(* CODESYS project intecreutilities.library
   DocFormat: reStructuredText
   Company: Intecre Ltd
   DefaultNamespace: Intecre.Utilities
   Title: Intecre.Utilities
   Placeholder: Intecre.Utilities
   Author: Mark Lazarides
   Description: 3.1.1.0 - adding long string list
      
      3.1.0.0 
      - Adding external logging injection
      3.0.0.0 
      - Renamed TNamedBase to T_NamedBase 
      - Added NONE level logging.
      - Logging is "NONE" by default.
      - Use something like "Intecre_Utilities.LogConfig.LogLevel := E_LogSeverity.Error; " to turn all on.
   Version: 3.1.1.0

Project tree, tasks and I/O mapping:
  libraries: Tc2_Math, * (Beckhoff Automation GmbH); Tc2_MDP, * (Beckhoff Automation GmbH); Tc2_Standard, * (Beckhoff Automation GmbH); Tc2_System, * (Beckhoff Automation GmbH); Tc2_Utilities, * (Beckhoff Automation GmbH); Tc3_Module, * (Beckhoff Automation GmbH)
  DUTs/
  GVLs/
    global variables CollectionParameters
    global variables LogConfig
    global variables Objects
    global variables StringsParams
  Project Information/
    function F_GetCompany [ST]
    function F_GetTitle [ST]
    function F_GetVersion [ST]
  System/
    function block T_Task [ST]: CycleCount, CyclesPerSecond, CycleTimeExceeded, CycleTimeInMs, CycleTimeInSecs, DateString, DateTimeFromDc, DateTimeString, DistributedClockTimeInMs, DistributedClockTimeInNs, DistributedClockTimeInSecs, Index, IsFirstScan, Name, TimeString, SetToThisTask
  Terminal Interfaces/
    Analogue Input EL3xxx/
      EL3058/
        data type stEL3058_Channel
        data type stEL3058_ChannelStatus
      EL3152/
        data type stEL3152_Channel
        data type stEL3152_ChannelStatus
      EL3318/
        data type stEL3318_Channel
        data type stEL3318_ChannelStatus
    EtherCAT Standard/
      data type stInfoData
      data type stWcState
    System EL9xxx/
      EL9410/
        data type stEL9410
      EL9576/
        data type stEL9576
        data type stEL9576_Status
  Utilities/
    Conversion/
      function CharIsNumber [ST]
      function CharIsNumberOrPeriod [ST]
      function TryStringToLreal [ST]
      function TryStringToUdint [ST]
      function TryStringToWord [ST]
    IPC Diagnostics/
      function block T_MdpReadCpuTemp [ST]: Busy, CpuTemp, Error, ErrorId, SetUpdateTimerValue
    Logger/
      data type E_LogSeverity
      function F_LogDebug [ST]
      function F_LogError [ST]
      function F_Logger [ST]
      function F_LogInfo [ST]
      function F_LogWarning [ST]
      function block FB_LogErrorEdge [ST]
      function block FB_LogInfoEdge [ST]
      function block FB_LogOnEdge [ST]
      function block FB_LogWarningEdge [ST]
      interface I_ExternalLogger: AddToLog
    Object Tracking/
      function F_DictionaryValuesCrc [ST]
      function block FB_Dictionary [ST]: AddItem, Clear, Contains, Count, Get, ReferenceToThis, Remove, TryGet, TryGetIndex, TryGetPartialKey
      function block FB_PointerList [ST]: AddItem, Clear, Contains, Count, FindIndex, GetIndex, RemoveIndex, TryGetIndex
      function block FB_StringList [ST]: AddItem, Clear, Contains, ContainsPartial, CopyList, CopyListAndClear, Count, FindIndex, FindIndexPartialKey, GetIndex, RemoveIndex, TryGetIndex
      function block FB_LongStringList [ST]: AddItem, Clear, Contains, ContainsPartial, CopyList, CopyListAndClear, Count, FindIndex, FindIndexPartialKey, GetIndex, RemoveIndex, TryGetIndex
      function block FB_TargList [ST]: AddItem, Clear, Contains, Count, FindIndex, GetIndex, RemoveIndex, TryGetIndex
      function block FB_UdintList [ST]: AddItem, Clear, Contains, Count, FindIndex, GetIndex, RemoveIndex, TryGetIndex
      global variables GVL_List
      data type ST_KeyReferencePair
    PI Controller/
      function block FB_I_Controller [ST]
      function block FB_P_Control [ST]
      function block FB_PI_Controller [ST]
    String/
      Large Concats/
        function F_ClearLarge [ST]
        function F_Concat3_Large [ST]
        function F_Concat4_Large [ST]
        function F_Concat5_Large [ST]
        function F_Concat6_Large [ST]
        function F_Concat7_Large [ST]
        function F_ConcatLarge [ST]
      data type LongString
      function F_Concat3 [ST]
      function F_Concat4 [ST]
      function F_Concat5 [ST]
      function F_Concat6 [ST]
      function F_Concat7 [ST]
      function F_StringToTarg [ST]
      function F_TargToString [ST]
    Testing/
      function block FB_Assert [ST]: FinishedTestingMsg, FloatsAreDifferent, FloatsAreEqual, IsFalse, IsTrue, StartTestingMsg
      function block T_TestBase [ST]: Done, DonePulse, nElapsedTimeInMs, Passed, Reset, Start, StartTimer, tElapsedTimeInMs
    Timers/
      function block T_Timer [ST]: ElapsedTime, ElapsedTimeInMs, Q_Off, Q_On, Q_PulseTrain, SetPeriod, Signal
    Write persistent/
      function block T_WritePersistentData [ST]: SetConfig
    function F_Gate [ST]
    function block T_NamedBase [ST]: InstanceName, LogDebug, LogError, LogInfo, LogWarning, setInstanceName
  Version/
    global variables Global_Version
  VISUs/
*)

// Terminal Interfaces/Analogue Input EL3xxx/EL3058/stEL3058_Channel
{attribute 'pack_mode' := '1'}
TYPE stEL3058_Channel :
STRUCT
	Status	AT %I* : stEL3058_ChannelStatus;
	Value 	AT %I* : WORD;
END_STRUCT
END_TYPE

// Terminal Interfaces/Analogue Input EL3xxx/EL3058/stEL3058_ChannelStatus
TYPE stEL3058_ChannelStatus :
STRUCT
	Underrange 	: BIT;
	Overrange	: BIT;
	Limit1_0	: BIT; // Value <= limit 1
	Limit1_1 	: BIT; // Value >= limit 1
	Limit2_0	: BIT; // Value <= limit 2
	Limit2_1	: BIT; // Value >= limit 2
	Error		: BIT; // TRUE when Over or under range.
	{attribute 'hide'}
	padding_0_7	: BIT;
	{attribute 'hide'}
	padding_1_0 : BIT;
	{attribute 'hide'}
	padding_1_1 : BIT;
	{attribute 'hide'}
	padding_1_2 : BIT;
	{attribute 'hide'}
	padding_1_3 : BIT;
	{attribute 'hide'}
	padding_1_4 : BIT;
	{attribute 'hide'}
	padding_1_5 : BIT;
	TxPDO_State : BIT; // TRUE when PDO NOT valid
	TxPDO_Toddle: BIT; // toggles when new value available
END_STRUCT
END_TYPE

// Terminal Interfaces/Analogue Input EL3xxx/EL3152/stEL3152_Channel
{attribute 'pack_mode' := '1'}
TYPE stEL3152_Channel:
STRUCT
	Status 	AT %I* : stEL3152_ChannelStatus;	
	Value 	AT %I* : WORD;  
END_STRUCT
END_TYPE;

// Terminal Interfaces/Analogue Input EL3xxx/EL3152/stEL3152_ChannelStatus
{attribute 'pack_mode' := '1'}
TYPE stEL3152_ChannelStatus:
STRUCT
	Underrange 	: BIT;
	Overrange 	: BIT;
	LT_Lim1 	: BIT; // Less Than Limit 1
	GT_Lim1 	: BIT; // Greater Than Limit 1
	LT_Lim2 	: BIT; // Less Than Limit 2
	GT_Lim2 	: BIT; // Greater Than Limit 2
	Error		: BIT;
	{attribute 'hide'}
	pack0_7		: BIT;	
	{attribute 'hide'}
	pack1_0		: BIT;
	{attribute 'hide'}
	pack1_1	 	: BIT;
	{attribute 'hide'}
	pack1_2	 	: BIT;
	{attribute 'hide'}
	pack1_3	 	: BIT;
	{attribute 'hide'}
	pack1_4	 	: BIT;
	SyncError	: BIT;
	TxPDOState	: BIT;
	TxPDOToggle : BIT;
END_STRUCT
END_TYPE;

// Terminal Interfaces/Analogue Input EL3xxx/EL3318/stEL3318_Channel
{attribute 'pack_mode' := '2'}
TYPE stEL3318_Channel:
STRUCT
	Status 	AT %I* : stEL3318_ChannelStatus;	 
	Value 	AT %I* : WORD;  
END_STRUCT
END_TYPE;

// Terminal Interfaces/Analogue Input EL3xxx/EL3318/stEL3318_ChannelStatus
{attribute 'pack_mode' := '1'}
TYPE stEL3318_ChannelStatus:
STRUCT
	Underrange 	: BIT;
	Overrange 	: BIT;
	{attribute 'hide'}
	pack_0_2	: BIT;
	{attribute 'hide'}
	pack_0_3	: BIT;
	{attribute 'hide'}
	pack_0_4	: BIT;
	{attribute 'hide'}
	pack_0_5	: BIT;
	Error		: BIT;
	{attribute 'hide'}	
	pack_0_7	: BIT;
	{attribute 'hide'}
	pack_1_0 	: BIT;
	{attribute 'hide'}
	pack_1_1 	: BIT;
	{attribute 'hide'}
	pack_1_2	: BIT;
	{attribute 'hide'}
	pack_1_3	: BIT;
	{attribute 'hide'}
	pack_1_4	: BIT;
	{attribute 'hide'}
	pack_1_5	: BIT;
	TxPDOState	: BIT;
	TxPDOToggle : BIT;

END_STRUCT
END_TYPE;

// Terminal Interfaces/EtherCAT Standard/stInfoData
TYPE stInfoData :
STRUCT
	State 		AT %I* : WORD;
	InfoData 	AT %I* : AMSADDR;
END_STRUCT
END_TYPE

// Terminal Interfaces/EtherCAT Standard/stWcState
TYPE stWcState :
STRUCT
	WcState		AT %I* : BOOL; // FALSE = data valid, TRUE = data not valid
	InputToggle	AT %I* : BOOL; // toggles every scan.
END_STRUCT
END_TYPE

// Terminal Interfaces/System EL9xxx/EL9410/stEL9410
TYPE stEL9410 :
STRUCT
	Us_Undervoltage  AT%I* : BIT; 
	Up_Undervoltage AT %I* : BIT; 
END_STRUCT
END_TYPE

// Terminal Interfaces/System EL9xxx/EL9576/stEL9576
{attribute 'pack_mode' := '1'}
TYPE stEL9576 :
STRUCT
	BCT_Inputs AT %I* : stEL9576_Status; 
END_STRUCT
END_TYPE;

// Terminal Interfaces/System EL9xxx/EL9576/stEL9576_Status
{attribute 'pack_mode' := '1'}
TYPE stEL9576_Status :
STRUCT
	TermOvertemp 	: BIT;
	I2T_Err 		: BIT;
	I2T_Warning 	: BIT; 
	Overvoltage 	: BIT; 
	Undervoltage 	: BIT; 
	ChopperOn 		: BIT;
	{attribute 'hide'}
	pack0_6		: BIT;
	{attribute 'hide'}
	pack0_7		: BIT;
	{attribute 'hide'}
	pack1_0		: BIT;
	{attribute 'hide'}
	pack1_1	 	: BIT;
	{attribute 'hide'}
	pack1_2	 	: BIT;
	{attribute 'hide'}
	pack1_3	 	: BIT;
	{attribute 'hide'}
	pack1_4	 	: BIT;
	{attribute 'hide'}
	pack1_5	 	: BIT;
	InputCycCnt_0	: BIT;
	InputCycCnt_1	: BIT;
	DcLinkVoltage	: UDINT;
	ResistorCurrent	: DINT;
	DutyCycle 		: USINT;
	I2T_LoadFactor 	: USINT;
END_STRUCT
END_TYPE;

// Utilities/Logger/E_LogSeverity
{attribute 'qualified_only'}
TYPE E_LogSeverity :
(
	Debug := 0,
	Info := ADSLOG_MSGTYPE_HINT,
	Warning := ADSLOG_MSGTYPE_WARN,
	Error := ADSLOG_MSGTYPE_ERROR,
	None := 1000
) DWORD;
END_TYPE

// Utilities/Object Tracking/ST_KeyReferencePair
TYPE ST_KeyReferencePair :
STRUCT
	Key : T_MaxString;
	Ref : T_Arg;
END_STRUCT
END_TYPE

// Utilities/String/LongString
TYPE LongString : STRING(StringsParams.MAX_STRING_LENGTH); END_TYPE // use StringsParams.MAX_STRING_LENGTH to adjust length

// GVLs/CollectionParameters
{attribute 'qualified_only'}
VAR_GLOBAL CONSTANT
	MAX_BYTE_SIZE : UDINT := 1000;
END_VAR

// GVLs/LogConfig
{attribute 'qualified_only'}
VAR_GLOBAL
	// set level to log. Lower log level includes higher levels i.e. info does warning and Error. 
	LogLevel : E_LogSeverity := E_LogSeverity.None; // Turn messages off by default
	ExternalLogger : I_ExternalLogger; // permit logging to something else
END_VAR

// GVLs/Objects
{attribute 'qualified_only'}
{attribute 'strict'}
VAR_GLOBAL 
	
END_VAR

// GVLs/StringsParams
{attribute 'qualified_only'}
VAR_GLOBAL CONSTANT
	MAX_STRING_LENGTH : UDINT := 300; // used for all string concats.
END_VAR

// Utilities/Object Tracking/GVL_List
{attribute 'qualified_only'}
VAR_GLOBAL CONSTANT
	LIST_SIZE : UINT := 100; // Number of list items.
END_VAR

// Version/Global_Version
{attribute 'TcGenerated'}
{attribute 'no-analysis'}
{attribute 'linkalways'}
// This function has been automatically generated from the project information.
VAR_GLOBAL CONSTANT
	{attribute 'const_non_replaced'}
	stLibVersion_Intecre_Utilities : ST_LibVersion := (iMajor := 3, iMinor := 1, iBuild := 1, iRevision := 0, sVersion := '3.1.1.0');
END_VAR

// Project Information/F_GetCompany
// This function has been automatically generated from the project information.
{attribute 'signature_flag' := '1073741824'}
{attribute 'TcGenerated'}
{attribute 'no-analysis'}
FUNCTION F_GetCompany : WSTRING
VAR_INPUT
	
END_VAR

F_GetCompany := "Intecre Ltd";

END_FUNCTION

// Project Information/F_GetTitle
// This function has been automatically generated from the project information.
{attribute 'signature_flag' := '1073741824'}
{attribute 'TcGenerated'}
{attribute 'no-analysis'}
FUNCTION F_GetTitle : WSTRING
VAR_INPUT
	
END_VAR

F_GetTitle := "Intecre.Utilities";

END_FUNCTION

// Project Information/F_GetVersion
// This function has been automatically generated from the project information.
{attribute 'signature_flag' := '1073741824'}
{attribute 'TcGenerated'}
{attribute 'no-analysis'}
FUNCTION F_GetVersion : ST_LibVersion
VAR_INPUT
	
END_VAR

F_GetVersion.iMajor := 3;
F_GetVersion.iMinor := 1;
F_GetVersion.iBuild := 1;
F_GetVersion.iRevision := 0;

END_FUNCTION

// System/T_Task
// Exposes _TaskInfo[x] information for the task index the object is instantied in.
//
// After declaration, each property can be directly accessed.
//
// Set the index using task.Index
FUNCTION_BLOCK T_Task // Simply exposes task information.
VAR
// Backing Properties
	_index : BYTE := 1;
	_cycleTimeInMs : LREAL;
	_isFirstScan : BOOL;
	_cycleTimeExceeded : BOOL;
	_name : STRING(63);
	_runTimeInMs : UDINT;
	_distributedClockTimeInMs : LINT;
	_distributedClockTimeInNs : LINT;

// FBs
	initialised : BOOL := FALSE;
	taskIndex : GETCURTASKINDEX;
	
END_VAR

VAR CONSTANT
	HUNDRED_NS_IN_MS : LINT := 10000;
	NS_IN_MS : LINT := 1000000;
END_VAR

// Number of task cycles executed.
PROPERTY PUBLIC CycleCount : UDINT
GET
cycleCount := TwinCAT_SystemInfoVarList._TaskInfo[_index].CycleCount;
END_GET
END_PROPERTY

// Configured cycles per second (1 / task time)
PROPERTY CyclesPerSecond : LREAL
GET
CyclesPerSecond := 1 / CycleTimeInSecs;
END_GET
END_PROPERTY

// Last cycle time exceeded
PROPERTY CycleTimeExceeded : BOOL
GET
_cycleTimeExceeded := TwinCAT_SystemInfoVarList._TaskInfo[_index].CycleTimeExceeded;
cycleTimeExceeded := _cycleTimeExceeded;
END_GET
END_PROPERTY

// Configured task cycle time in ms
PROPERTY CycleTimeInMs : LREAL
GET
_cycleTimeInMs := TwinCAT_SystemInfoVarList._TaskInfo[_index].CycleTime / LINT_TO_UDINT(HUNDRED_NS_IN_MS); // CycleTime expressed in 100ns units.
cycleTimeInMs := _cycleTimeInMs;
END_GET
END_PROPERTY

// Configured task cycle time in seconds
PROPERTY CycleTimeInSecs : LREAL
GET
CycleTimeInSecs:= CycleTimeInMs / 1000;
END_GET
END_PROPERTY

PROPERTY DateString : STRING
GET
VAR
	temp : STRING;
END_VAR
// remove the trailing time: 2018-07-30_09-23-47
temp := DELETE( TO_STRING( DateTimeString ), 9,11 );

// 2018-07-30
DateString :=  temp;
END_GET
END_PROPERTY

PROPERTY DateTimeFromDc : DATE_AND_TIME
GET
DateTimeFromDc := LINT_TO_DT( TO_LINT( DT#2000-1-1-00:00 ) + TwinCAT_SystemInfoVarList._TaskInfo[_index].DcTaskTime / 1000000000 );
END_GET
END_PROPERTY

PROPERTY DateTimeString : STRING
GET
VAR
	temp : STRING;
END_VAR
// remove the leading DT# : DT#2018-07-30-09:23:47
temp := DELETE( TO_STRING( DateTimeFromDc ), 3, 1 );
// add underscore between datae and time 2018-07-30-09:23:47
temp := REPLACE( temp, '_', 1, 11 );
// replace the colons with dashes 2018-07-30_09:23:47
temp := REPLACE( REPLACE( temp, '-', 1, 14 ), '-', 1, 17 );

// 2018-07-30_09-23-47
DateTimeString :=  temp;
END_GET
END_PROPERTY

//Distributed clock time in milliseconds.
PROPERTY PUBLIC DistributedClockTimeInMs : LINT
GET
_distributedClockTimeInMs := TwinCAT_SystemInfoVarList._TaskInfo[_index].DcTaskTime / NS_IN_MS; // CycleTime expressed ns.
DistributedClockTimeInMs := _distributedClockTimeInMs;
END_GET
END_PROPERTY

//Distributed clock time in nanoseconds.
PROPERTY PUBLIC DistributedClockTimeInNs : LINT
GET
_distributedClockTimeInNs := TwinCAT_SystemInfoVarList._TaskInfo[_index].DcTaskTime; // CycleTime expressed ns.
DistributedClockTimeInNs := _distributedClockTimeInNs;
END_GET
END_PROPERTY

//Distributed clock time in milliseconds.
PROPERTY PUBLIC DistributedClockTimeInSecs : LINT
GET
DistributedClockTimeInSecs := DistributedClockTimeInMs / 1000;
END_GET
END_PROPERTY

//Get/Set the task for the infomration required. Can use "SetToThisTask()" to set to local task.
PROPERTY PUBLIC Index : BYTE
GET
PUBLIC
Index := _index;
END_GET
SET
PUBLIC
_index := Index;
END_SET
END_PROPERTY

PROPERTY IsFirstScan : BOOL
GET
_isFirstScan := TwinCAT_SystemInfoVarList._TaskInfo[_index].FirstCycle;
IsFirstScan := _isFirstScan;
END_GET
END_PROPERTY

{attribute 'monitoring' := 'call'}
PROPERTY Name : STRING(63)
GET
_name := TwinCAT_SystemInfoVarList._TaskInfo[_index].TaskName;
Name := _name;
END_GET
END_PROPERTY

PROPERTY TimeString : STRING
GET
VAR
	temp : STRING;
END_VAR
// remove the leading date 2018-07-30_09-23-47
temp := DELETE( TO_STRING( DateTimeString ), 11, 1 );

// 09-23-47
TimeString :=  temp;
END_GET
END_PROPERTY

//set the task object to this task
METHOD PUBLIC SetToThisTask : BOOL
VAR
	curTask : GETCURTASKINDEX;
END_VAR
curTask();
Index := curTask.index;
END_METHOD

END_FUNCTION_BLOCK

// Utilities/Conversion/CharIsNumber
FUNCTION CharIsNumber : BOOL
VAR_INPUT
	bChar : BYTE; // char to check
END_VAR

// check bChar is in numbr range of ascii
CharIsNumber := (bChar >= 48 AND bChar <=57);

END_FUNCTION

// Utilities/Conversion/CharIsNumberOrPeriod
FUNCTION CharIsNumberOrPeriod : BOOL
VAR_INPUT
	bChar : BYTE; // char to check
END_VAR

// check is bChar in number range of ascii, or a period (full-stop).
CharIsNumberOrPeriod := CharIsNumber( bChar ) OR_ELSE (bChar = 46);

END_FUNCTION

// Utilities/Conversion/TryStringToLreal
// Returns TRUE if possible. sVal will hold value if passes.
FUNCTION TryStringToLreal : BOOL 
VAR_INPUT
	sStringToParse : STRING; // String to try
END_VAR
VAR_IN_OUT
	sVal : LREAL; // 0.0 (zero) if fails, parsed value if passes.
END_VAR
VAR
	i : INT;
	n : INT; // position of full stop (if at all).
	intPart : DINT; // integer part of the number.
	decPart : UDINT; // decimal part of the number.
	decPartAsLreal : LREAL;
	decimalPlaces : INT; // number of dps.
	isMinus : BOOL;
END_VAR

IF LEN(sStringToParse) > 0 THEN

	FOR i := 0 TO LEN(sStringToParse) - 1 DO	
		
		IF i = 0 AND_THEN sStringToParse[i] = 45 THEN // accept "minus" sign for first digit
			isMinus := TRUE;
		ELSIF i = 1 AND isMinus THEN // if first char is "-", second must be digit.
			IF NOT CharIsNumberOrPeriod( sStringToParse[i] ) THEN
				sVal := 0;
				RETURN;
			END_IF
		ELSIF NOT CharIsNumberOrPeriod( sStringToParse[i] ) THEN
			sVal := 0;
			RETURN;
		END_IF	
	END_FOR
	
	n := FIND(sStringToParse, '.');
	
	IF n > 0 THEN // full stop is in the string.
		// get integer part.
		intPart := STRING_TO_DINT(LEFT(sStringToParse, n - 1));
		decimalPlaces := LEN(sStringToParse) - n;
		// get decimal part as integer.
		decPart := STRING_TO_UDINT( RIGHT(sStringToParse, decimalPlaces) );
		// convert to LREAL, includng rolling decimal places.
		decPartAsLreal := UDINT_TO_LREAL(decPart)/EXPT(10,decimalPlaces);
		// handle sign change.
		IF isMinus THEN
			decPartAsLreal := decPartAsLreal * -1;
		END_IF
		
		//combine them
		sVal := DINT_TO_LREAL(intPart);
		sVal := sVal + decPartAsLreal;
	ELSE
		sVal := STRING_TO_LREAL(sStringToParse);
	END_IF
	
	TryStringToLreal := TRUE;
	
END_IF

END_FUNCTION

// Utilities/Conversion/TryStringToUdint
// Returns TRUE if possible. sVal will hold value if passes.
FUNCTION TryStringToUdint : BOOL 
VAR_INPUT
	sStringToParse : STRING; // String to try
END_VAR
VAR_IN_OUT
	sVal : UDINT; // 0 (zero) if fails, parsed value if passes.
END_VAR
VAR
	i : INT;
END_VAR

IF LEN(sStringToParse) > 0 THEN

	FOR i := 0 TO LEN(sStringToParse) - 1 DO		
		IF NOT CharIsNumber( sStringToParse[i] ) THEN
			sVal := 0;
			RETURN;
		END_IF	
	END_FOR
	
	sVal := STRING_TO_UDINT( sStringToParse );
	TryStringToUdint := TRUE;
	
END_IF

END_FUNCTION

// Utilities/Conversion/TryStringToWord
// Returns TRUE if possible. sVal will hold value if passes. 
//
// Internally this casts to Udint, then checks value is <= MAX_WORD
FUNCTION TryStringToWord : BOOL 
VAR_INPUT
	sStringToParse : STRING; // String to try
END_VAR
VAR_IN_OUT
	sVal : WORD; // 0 (zero) if fails, parsed value if passes.
END_VAR
VAR
	u : UDINT;
END_VAR

// check parsing to UDINT possible, then validate size of word.
IF TryStringToUdint(sStringToParse, u) THEN
	// check within WORD size.
	IF UDINT_TO_WORD(u) <= 65535 THEN
		sVal := STRING_TO_WORD( sStringToParse );
		TryStringToWord := TRUE;
	END_IF
	
END_IF

END_FUNCTION

// Utilities/IPC Diagnostics/T_MdpReadCpuTemp
/// cyclically reads the  cpu temp at specified update period. Default is 500ms.
{attribute 'contains_implicit_enum'}
FUNCTION_BLOCK T_MdpReadCpuTemp
VAR
	/// local read                
	amsNetId: STRING := '';
	mdpAddr: ST_MDP_Addr;
	updateTimer: TON := (PT := TIME#500ms);
	readMdpElement: FB_MDP_ReadElement;
	/// returned from MDP read element 
	rawData: UINT;
	_cpuTemp: INT;
	{attribute 'implicit_enum_type' := ''}
	state:(
		mrctInit  := 0,     // initiate state machine (set parameters)
		mrctReadCpuTemp,
		mrctWaitForReadComplete,
		mrctProcessCpuTemp
	);   
END_VAR
VAR CONSTANT
	/// from IPC Diagnostics Manual V1.8, p63 
	CPU_PROPERTIES_TABLE_NUMBER: BYTE := 1;
	/// from IPC Diagnostics Manual V1.8, p63 
	CPU_TEMP_SUB_INDEX_OF_CPU_PROPS_TABLE: BYTE := 3;
END_VAR

CASE state OF

	mrctInit : 
		
		// timer starts the read process.
		state := 
			SEL ( updateTimer.Q, state, mrctReadCpuTemp );
		
	mrctReadCpuTemp :    
      
		state := mrctWaitForReadComplete;  
            
	mrctWaitForReadComplete :    

		IF NOT readMdpElement.bBusy THEN
			
			state := mrctProcessCpuTemp;
			
		END_IF
	
	mrctProcessCpuTemp :              

		IF NOT readMdpElement.bError THEN
			MEMCPY( ADR( _cpuTemp ), ADR( rawData ), SIZEOF( rawData ) );
			
		END_IF
		
		state    := mrctInit; 
		
ELSE
	
    state := mrctInit;   
	 
END_CASE 

updateTimer( 
	IN := state = mrctInit
);
		
mdpAddr.nArea := INT_TO_BYTE(eMDP_Area_ConfigArea); 
mdpAddr.nTableId := CPU_PROPERTIES_TABLE_NUMBER;            
mdpAddr.nSubIdx := CPU_TEMP_SUB_INDEX_OF_CPU_PROPS_TABLE;   

readMdpElement(
	bExecute	:= state = mrctReadCpuTemp,               
	eModuleType	:= E_MDP_ModuleType.eMDP_ModT_CPU,         
	stMDP_Addr := mdpAddr,          
	iModIdx := 0,                   
	pDstBuf := ADR(rawData),         
	cbDstBufLen := SIZEOF(rawData),  
	sAmsNetId := amsNetId,        
);

{attribute 'monitoring' := 'variable'}
PROPERTY Busy : BOOL
GET
Busy := state <> mrctInit;
END_GET
END_PROPERTY

{attribute 'monitoring' := 'call'}
PROPERTY CpuTemp : INT
GET
CpuTemp := THIS^._cpuTemp;
END_GET
END_PROPERTY

{attribute 'monitoring' := 'variable'}
PROPERTY Error : BOOL
GET
Error := NOT Busy AND readMdpElement.bError;
END_GET
END_PROPERTY

{attribute 'monitoring' := 'variable'}
PROPERTY ErrorId : UDINT
GET
ErrorId := SEL( Busy, readMdpElement.nErrID, 0 );
END_GET
END_PROPERTY

METHOD SetUpdateTimerValue 
VAR_INPUT	
	UpdatePeriod: TIME;
END_VAR
IF UpdatePeriod > T#1MS THEN
	THIS^.updateTimer.PT := UpdatePeriod;
END_IF
END_METHOD

END_FUNCTION_BLOCK

// Utilities/Logger/F_LogDebug
FUNCTION F_LogDebug : STRING;
VAR_INPUT
	Message : T_MaxString;
END_VAR

F_LogDebug := 
	F_Logger( 
		E_LogSeverity.Debug, 
		CONCAT( 'DEBUG ' , Message ) 
	);

END_FUNCTION

// Utilities/Logger/F_Logger
FUNCTION F_Logger : STRING;
VAR_INPUT
	LogSeverity : E_LogSeverity;
	Message : T_MaxString;
END_VAR

IF ( LogSeverity < E_LogSeverity.None ) 
	AND_THEN ( LogSeverity >= LogConfig.LogLevel ) THEN
	
	ADSLOGSTR(LogSeverity OR ADSLOG_MSGTYPE_LOG, Message, '');
	F_Logger := Message;
	
	IF LogConfig.ExternalLogger <> 0 THEN
		LogConfig.ExternalLogger.AddToLog( Message, LogSeverity );
	END_IF
	
END_IF

END_FUNCTION

// Utilities/Logger/F_LogError
FUNCTION F_LogError : STRING;
VAR_INPUT
	Message : T_MaxString;
END_VAR

F_LogError := F_Logger(ADSLOG_MSGTYPE_ERROR, Message);

END_FUNCTION

// Utilities/Logger/F_LogInfo
FUNCTION F_LogInfo : STRING;
VAR_INPUT
	Message : T_MaxString;
END_VAR

F_LogInfo := F_Logger(ADSLOG_MSGTYPE_HINT, Message);

END_FUNCTION

// Utilities/Logger/F_LogWarning
FUNCTION F_LogWarning : STRING;
VAR_INPUT
	Message : T_MaxString;
END_VAR

F_LogWarning := F_Logger(ADSLOG_MSGTYPE_WARN, Message);

END_FUNCTION

// Utilities/Logger/FB_LogErrorEdge
FUNCTION_BLOCK FB_LogErrorEdge
VAR_INPUT
	Event : BOOL; // Event flag
	Message : T_MaxString; // Log message
	EventFallingEdge : BOOL := FALSE; // Defined which edge: FALSE = rising TRUE = falling, 
END_VAR
VAR_OUTPUT
	Q : BOOL;
END_VAR
VAR
	fbLogEdge : FB_LogOnEdge;
END_VAR

fbLogEdge(
	Event:= Event, 
	Message:= Message, 
	LogSeverity:= E_LogSeverity.Error, 
	EventFallingEdge:= EventFallingEdge,
	Q => Q
);

END_FUNCTION_BLOCK

// Utilities/Logger/FB_LogOnEdge
FUNCTION_BLOCK FB_LogOnEdge
VAR_INPUT
	Event : BOOL; // look for edge here to log.
	Message : T_MaxString; // message
	LogSeverity : E_LogSeverity; // severity
	EventFallingEdge : BOOL := FALSE; // TRUE for falling edge, FALSE for rising edge.
END_VAR
VAR_OUTPUT
	Q : BOOL;
END_VAR
VAR
	rt : R_TRIG;
	ft : F_TRIG;
END_VAR
VAR_TEMP
	logNow : BOOL;
END_VAR

rt(CLK := Event);
ft(CLK := Event);

Q := SEL(EventFallingEdge, rt.Q, ft.Q);

IF Q THEN
	
	CASE LogSeverity OF
		
		E_LogSeverity.Info : F_LogInfo(Message);
			
		E_LogSeverity.Warning :	F_LogWarning(Message);
			
		E_LogSeverity.Error : F_LogError(Message);
	ELSE 
		
		F_LogError(
			CONCAT(
				'Error in FB_LogOnEdge, Logseverity incorrect. Log Message for event is : ', 
				Message
			)
		);
		
	END_CASE
	
END_IF

END_FUNCTION_BLOCK

// Utilities/Logger/FB_LogInfoEdge
FUNCTION_BLOCK FB_LogInfoEdge
VAR_INPUT
	Event : BOOL; // Event flag
	Message : T_MaxString; // Log message
	EventFallingEdge : BOOL := FALSE; // Defined which edge: FALSE = rising TRUE = falling, 
END_VAR
VAR_OUTPUT
	Q : BOOL;
END_VAR
VAR
	fbLogEdge : FB_LogOnEdge;
END_VAR

fbLogEdge(
	Event:= Event, 
	Message:= Message, 
	LogSeverity:= E_LogSeverity.Info, 
	EventFallingEdge:= EventFallingEdge,
	Q => Q
);

END_FUNCTION_BLOCK

// Utilities/Logger/FB_LogWarningEdge
FUNCTION_BLOCK FB_LogWarningEdge
VAR_INPUT
	Event : BOOL; // Event flag
	Message : T_MaxString; // Log message
	EventFallingEdge : BOOL := FALSE; // Defined which edge: FALSE = rising TRUE = falling, 
END_VAR
VAR_OUTPUT
	Q : BOOL;
END_VAR
VAR
	fbLogEdge : FB_LogOnEdge;
END_VAR

fbLogEdge(
	Event:= Event, 
	Message:= Message, 
	LogSeverity:= E_LogSeverity.Warning, 
	EventFallingEdge:= EventFallingEdge,
	Q => Q
);

END_FUNCTION_BLOCK

// Utilities/Logger/I_ExternalLogger
INTERFACE I_ExternalLogger

METHOD AddToLog
VAR_IN_OUT
	Message : T_MaxString;
END_VAR
VAR_INPUT
	LogSeverity : E_LogSeverity;
END_VAR
END_METHOD

END_INTERFACE

// Utilities/Object Tracking/F_DictionaryValuesCrc
// Return CRC of the values stored in the dictionary.
FUNCTION F_DictionaryValuesCrc : WORD
VAR_IN_OUT
	Dictionary : FB_Dictionary;
END_VAR
VAR
	i : UDINT;
	sKey : T_MaxString;
	tValue : T_Arg;
END_VAR

IF Dictionary.Count > 0 THEN
	
	IF NOT Dictionary.TryGetIndex(Index := 0, Key := sKey, Value := tValue) THEN
		RETURN;
	ELSE
		F_DictionaryValuesCrc := F_DATA_TO_CRC16_CCITT(
			pData := tValue.pData,
			cbData := tValue.cbLen,
			crc := 16#FFFF // First pass needs the seed.
			);
	END_IF
	
END_IF

FOR i := 1 TO (Dictionary.Count -1) DO
	
	IF NOT Dictionary.TryGetIndex(Index := 0, Key := sKey, Value := tValue) THEN
		F_DictionaryValuesCrc := 16#0000;
		RETURN;
	ELSE
		F_DictionaryValuesCrc := F_DATA_TO_CRC16_CCITT(
			pData := tValue.pData,
			cbData := tValue.cbLen,
			crc := F_DictionaryValuesCrc // iteratively pass in CRC.
			);
	END_IF
	
END_FOR

END_FUNCTION

// Utilities/Object Tracking/FB_Dictionary
FUNCTION_BLOCK FB_Dictionary EXTENDS T_NamedBase
VAR
	Keys : FB_StringList;
	Values : FB_TargList;
END_VAR

// Add item to list. TRUE if successful. 
METHOD PUBLIC AddItem : BOOL
VAR_INPUT
	Key : T_MaxString; // item key to add.
	Value : T_Arg;
END_VAR
IF Keys.Count <> Values.Count THEN
	LogWarning('Missmatch keys and values count. Clearing dictionary.');
	THIS^.Clear();
	RETURN;
END_IF
IF Keys.Count = GVL_List.LIST_SIZE THEN
	F_LogWarning(
		CONCAT(InstanceName, 'Dictionary is full.')
	);
	RETURN;
END_IF
IF Key = '' THEN
	LogWarning('key is null.');
	RETURN;
END_IF
IF Contains( Key )  THEN
	LogWarning('Key already exists in dictionary.');
	RETURN;
END_IF

IF Value.cbLen <= 0 THEN
	LogWarning('Value has no length.');
	RETURN;
END_IF

// Add the key.
IF NOT Keys.AddItem( Key ) THEN
	F_LogWarning(
		CONCAT(InstanceName, ' error adding key.')
	);
	RETURN;
END_IF
// add the value.
IF NOT Values.AddItem( Value ) THEN // if this fails, remove the key.
	LogWarning('Error adding value.');
	Keys.RemoveIndex( 
		INT_TO_UDINT( Keys.FindIndex( Key ) )
	);
	RETURN;
END_IF

AddItem := TRUE;
END_METHOD

// Removes all list items
METHOD PUBLIC Clear
Keys.Clear();
Values.Clear();
END_METHOD

// TRUE if Item is in FB_List.
METHOD PUBLIC Contains : BOOL
VAR_INPUT
	Key : T_MaxString; // Item to check.
END_VAR
VAR
	i : UINT := 0;
END_VAR
Contains := Keys.Contains ( Key );
END_METHOD

{attribute 'monitoring' := 'call'}
// Number of items in list.
PROPERTY PUBLIC Count : UDINT
GET
Count := Keys.Count;
END_GET
END_PROPERTY

// Return item in dictionary base on key.
METHOD PUBLIC Get : T_Arg
VAR_INPUT
	Key : T_MaxString;
END_VAR
THIS^.TryGet(Key, Get);
END_METHOD

PROPERTY PUBLIC ReferenceToThis : REFERENCE TO FB_Dictionary
GET
ReferenceToThis REF= THIS^;
END_GET
END_PROPERTY

//Remove the specified index. Shuffle remaining so list is intact.
METHOD PUBLIC Remove : BOOL
VAR_INPUT
	Key : T_MaxString;
END_VAR
IF Keys.Contains( Key ) THEN // invalid index request.
	LogWarning('Cannot remove key as not in dictionary.');
	RETURN;
END_IF

Values.RemoveIndex(
	INT_TO_UDINT( Keys.FindIndex( Key ) ) 
);

Keys.RemoveIndex( 
	INT_TO_UDINT( Keys.FindIndex( Key ) ) 
);

Remove := TRUE;
END_METHOD

// TRUE if successful and list item in sItem
METHOD PUBLIC TryGet : BOOL
VAR_INPUT
	Key : T_MaxString;
END_VAR
VAR_IN_OUT
	Value : T_Arg;
END_VAR
IF Keys.Contains( Key ) THEN
	Value := Values.GetIndex( 
				INT_TO_UDINT( Keys.FindIndex( Key ) ) 
			);
	TryGet := TRUE;
END_IF
END_METHOD

// TRUE if successful and list item in sItem
METHOD PUBLIC TryGetIndex : BOOL
VAR_INPUT
	Index : UDINT;
END_VAR
VAR_IN_OUT
	Key : T_MaxString;
	Value : T_Arg;
END_VAR
IF Index < Keys.Count THEN
	Key := Keys.GetIndex( Index );
	Value := Values.GetIndex( Index );
	TryGetIndex := TRUE;
END_IF
END_METHOD

// TRUE if successful. Returns value associated with first key that provides partial match
METHOD PUBLIC TryGetPartialKey : BOOL
VAR_IN_OUT CONSTANT
	PartialKey : T_MaxString;
END_VAR
VAR_IN_OUT
	Value : T_Arg;
END_VAR
IF Keys.ContainsPartial( PartialKey ) THEN
	Value := Values.GetIndex( 
				INT_TO_UDINT( Keys.FindIndexPartialKey( PartialKey ) ) 
			);
	TryGetPartialKey := TRUE;
END_IF
END_METHOD

END_FUNCTION_BLOCK

// Utilities/T_NamedBase
{attribute 'reflection'}
FUNCTION_BLOCK T_NamedBase
VAR
	{attribute 'instance-path'}
    {attribute 'no_init'}
	name : STRING;
	_instanceName : STRING; // name minus project name etc.
	_instanceSet : BOOL;
END_VAR

PROPERTY FINAL InstanceName : T_MaxString;
GET
IF NOT _instanceSet THEN
	setInstanceName();
END_IF

InstanceName := _instanceName;
END_GET
END_PROPERTY

METHOD LogDebug
VAR_INPUT
	Msg : T_MaxString;
END_VAR
F_LogDebug(
	F_Concat3(InstanceName , ': ', Msg)
);
END_METHOD

METHOD LogError
VAR_INPUT
	Msg : T_MaxString;
END_VAR
F_LogError(
	F_Concat3(InstanceName , ': ', Msg)
);
END_METHOD

METHOD LogInfo
VAR_INPUT
	Msg : T_MaxString;
END_VAR
F_LogInfo(
	F_Concat3(InstanceName , ': ', Msg)
);
END_METHOD

METHOD LogWarning
VAR_INPUT
	Msg : T_MaxString;
END_VAR
F_LogWarning(
	F_Concat3(InstanceName , ': ', Msg)
);
END_METHOD

METHOD PRIVATE setInstanceName 
VAR
	charsToDeleteFromPath : INT;
END_VAR
// format is  Solution_Name.ProjectName.FirstDeclaredPOU.etc.etc... 

//Remove Solution_Name
charsToDeleteFromPath := FIND( name, '.' );
_instanceName := DELETE( name, charsToDeleteFromPath, 1 );

//Remove ProjectName
charsToDeleteFromPath := FIND( _instanceName, '.' );

//gives us just "FirstDeclaredPOU.etc.etc..." from above.
_instanceName := DELETE( _instanceName, charsToDeleteFromPath, 1 );

_instanceSet := TRUE;
END_METHOD

END_FUNCTION_BLOCK

// Utilities/String/F_Concat3
FUNCTION F_Concat3 : T_MaxString
VAR_INPUT
	StringOne 	: STRING;
	StringTwo	: STRING;
	StringThree	: STRING;
END_VAR
VAR
	response : T_MaxString;
END_VAR

response := CONCAT( StringOne, StringTwo );
response := CONCAT( response, StringThree );
F_Concat3 := response;

END_FUNCTION

// Utilities/Object Tracking/FB_StringList
// List of Strings.
FUNCTION_BLOCK FB_StringList
VAR
	List : ARRAY[ 0 .. GVL_List.LIST_SIZE - 1 ] OF T_MaxString; // hold list
	_Count : UDINT := 0; // number of items.
END_VAR

// Add item to list. TRUE if successful. 
METHOD PUBLIC AddItem : BOOL
VAR_INPUT
	Item : T_MaxString; // item to add.
END_VAR
IF _Count < GVL_List.LIST_SIZE THEN
	List[_Count] := Item; // list is zero indexed, so number of items points at next free space.
	_Count := _Count + 1; 
	AddItem := TRUE;
END_IF
END_METHOD

// Removes all list items
METHOD PUBLIC Clear
MEMSET(ADR(List[0]), 0, SIZEOF(List));
_Count := 0;
END_METHOD

// TRUE if Item is in FB_List.
METHOD PUBLIC Contains : BOOL
VAR_INPUT
	Item : T_MaxString; // Item to check.
END_VAR
Contains := FindIndex(Item) >= 0;
END_METHOD

// TRUE if supplied key part is in any entry
METHOD PUBLIC ContainsPartial : BOOL
VAR_INPUT
	PartialItem : T_MaxString;
END_VAR
ContainsPartial := FindIndexPartialKey(PartialItem) >= 0;
END_METHOD

METHOD CopyList
VAR_IN_OUT
	ListToCopyTo : ARRAY[ 0 .. GVL_List.LIST_SIZE - 1 ] OF T_MaxString; // hold list
END_VAR
ListToCopyTo := THIS^.List;
END_METHOD

METHOD CopyListAndClear
VAR_IN_OUT
	ListToCopyTo : ARRAY[ 0 .. GVL_List.LIST_SIZE - 1 ] OF T_MaxString; // hold list
END_VAR
THIS^.CopyList( ListToCopyTo );
THIS^.Clear();
END_METHOD

{attribute 'monitoring' := 'call'}
// Number of items in list.
PROPERTY PUBLIC Count : UDINT
GET
Count := _Count;
END_GET
END_PROPERTY

METHOD PUBLIC FindIndex : INT
VAR_INPUT
	Item : T_MaxString; // Item to check.
END_VAR
VAR
	i : UINT := 0;
END_VAR
FindIndex := -1;
i := 0;
WHILE ( (FindIndex < 0) AND (i < _Count) ) DO
	
	FindIndex := SEL(Item = List[i], FindIndex, TO_INT(i) ); // if it matches, return the position.
	i := i + 1;
	
END_WHILE
END_METHOD

// Find first index where list entry contains supplied key.
METHOD PUBLIC FindIndexPartialKey : INT
VAR_INPUT
	PartialKey : T_MaxString; // Item to check.
END_VAR
VAR
	i : UINT := 0;
END_VAR
FindIndexPartialKey := -1;
i := 0;
WHILE ( (FindIndexPartialKey < 0) AND (i < _Count) ) DO
	
	IF FIND(List[i],PartialKey) > 0 THEN
		FindIndexPartialKey := TO_INT(i);
	END_IF

	i := i + 1;
	
END_WHILE
END_METHOD

// Return item in list at index position. Returns empty string if invalid index.
METHOD PUBLIC GetIndex : T_MaxString
VAR_INPUT
	Index : UDINT;
END_VAR
THIS^.TryGetIndex(Index,  GetIndex);
END_METHOD

//Remove the specified index. Shuffle remaining so list is intact.
METHOD PUBLIC RemoveIndex : BOOL
VAR_INPUT
	Index : UDINT;
END_VAR
IF Index >= _Count THEN // invalid index request.
	RETURN;
END_IF

IF Index < _Count - 1 THEN // If Index = _Count -1, last two lines sufficient.

	MEMMOVE( 
		destAddr := ADR( List[Index] ), 
		srcAddr := ADR( List[Index + 1] ), 
		n := SIZEOF(List[0]) * (_Count - Index - 1)
	);
	
END_IF

RemoveIndex := TRUE;

List[_Count - 1] := ''; // default the "old" end of the list.
_Count := _Count - 1; // reduce count.
END_METHOD

// TRUE if successful and list item in sItem
METHOD PUBLIC TryGetIndex : BOOL
VAR_INPUT
	Index : UDINT;
END_VAR
VAR_IN_OUT
	Item : T_MaxString;
END_VAR
IF Index < _Count THEN
	TryGetIndex := TRUE;
	Item := List[Index];
END_IF
END_METHOD

END_FUNCTION_BLOCK

// Utilities/Object Tracking/FB_TargList
// List of Strings.
FUNCTION_BLOCK FB_TargList
VAR
	List : ARRAY[ 0 .. GVL_List.LIST_SIZE - 1 ] OF T_Arg; // hold list
	_Count : UDINT := 0; // number of items.
END_VAR

// Add item to list. TRUE if successful. 
METHOD PUBLIC AddItem : BOOL
VAR_INPUT
	Item : T_Arg; // item to add.
END_VAR
IF _Count < GVL_List.LIST_SIZE THEN
	List[_Count] := Item; // list is zero indexed, so number of items points at next free space.
	_Count := _Count + 1; 
	AddItem := TRUE;
END_IF
END_METHOD

// Removes all list items
METHOD PUBLIC Clear
MEMSET(ADR(List[0]), 0, SIZEOF(List));
_Count := 0;
END_METHOD

// TRUE if Item is in FB_List.
METHOD PUBLIC Contains : BOOL
VAR_INPUT
	Item : T_Arg; // Item to check.
END_VAR
Contains := FindIndex(Item) >= 0;
END_METHOD

{attribute 'monitoring' := 'call'}
// Number of items in list.
PROPERTY PUBLIC Count : UDINT
GET
Count := _Count;
END_GET
END_PROPERTY

METHOD PUBLIC FindIndex : INT
VAR_INPUT
	Item : T_Arg; // Item to check.
END_VAR
VAR
	i : UINT := 0;
END_VAR
FindIndex := -1;
i := 0;
WHILE ( (FindIndex < 0) AND (i < _Count) ) DO
	
	FindIndex := SEL(F_ARGCMP(TRUE, Item, List[i]) = 0, FindIndex, TO_INT(i) ); // if it matches, return the position.
	i := i + 1;
	
END_WHILE
END_METHOD

// Return item in list at index position. Returns empty string if invalid index.
METHOD PUBLIC GetIndex : T_Arg
VAR_INPUT
	Index : UDINT;
END_VAR
THIS^.TryGetIndex(Index,  GetIndex);
END_METHOD

//Remove the specified index. Shuffle remaining so list is intact.
METHOD PUBLIC RemoveIndex : BOOL
VAR_INPUT
	Index : UDINT;
END_VAR
IF Index >= _Count THEN // invalid index request.
	RETURN;
END_IF

IF Index < _Count - 1 THEN // If Index = _Count -1, last two lines sufficient.

	MEMMOVE( 
		destAddr := ADR( List[Index] ), 
		srcAddr := ADR( List[Index + 1] ), 
		n := SIZEOF(List[0]) * (_Count - Index - 1)
	);
	
END_IF

RemoveIndex := TRUE;
MEMSET(ADR(List[_Count - 1]), 0, SIZEOF(T_Arg));
_Count := _Count - 1; // reduce count.
END_METHOD

// TRUE if successful and list item in sItem
METHOD PUBLIC TryGetIndex : BOOL
VAR_INPUT
	Index : UDINT;
END_VAR
VAR_IN_OUT
	Item : T_Arg;
END_VAR
IF Index < _Count THEN
	TryGetIndex := TRUE;
	Item := List[Index];
END_IF
END_METHOD

END_FUNCTION_BLOCK

// Utilities/Object Tracking/FB_PointerList
// List of UDINTs.
FUNCTION_BLOCK FB_PointerList
VAR
	List : ARRAY[ 0 .. GVL_List.LIST_SIZE - 1 ] OF PVOID; // hold list
	_Count : UDINT := 0; // number of items.
END_VAR

// Add item to list. TRUE if successful. 
METHOD PUBLIC AddItem : BOOL
VAR_INPUT
	Item : PVOID; // item to add.
END_VAR
IF _Count < GVL_List.LIST_SIZE THEN
	List[_Count] := Item; // list is zero indexed, so number of items points at next free space.
	_Count := _Count + 1; 
	AddItem := TRUE;
END_IF
END_METHOD

// Removes all list items
METHOD PUBLIC Clear
MEMSET(ADR(List[0]), 0, SIZEOF(List));
_Count := 0;
END_METHOD

// TRUE if sItem is in FB_List.
METHOD PUBLIC Contains : BOOL
VAR_INPUT
	Item : PVOID; // Item to check.
END_VAR
Contains := FindIndex(Item) >= 0;
END_METHOD

{attribute 'monitoring' := 'call'}
// Number of items in list.
PROPERTY PUBLIC Count : UDINT
GET
Count := _Count;
END_GET
END_PROPERTY

METHOD PUBLIC FindIndex : INT
VAR_INPUT
	Item : PVOID; // Item to check.
END_VAR
VAR
	i : UINT := 0;
END_VAR
FindIndex := -1;
i := 0;
WHILE ( (FindIndex < 0) AND (i < _Count) ) DO
	
	FindIndex := SEL(Item = List[i], FindIndex, TO_INT(i) ); // if it matches, return the position.
	i := i + 1;
	
END_WHILE
END_METHOD

// Return item in list at index position. Returns empty string if invalid index.
METHOD PUBLIC GetIndex : PVOID
VAR_INPUT
	Index : PVOID;
END_VAR
THIS^.TryGetIndex(Index,  GetIndex);
END_METHOD

//Remove the specified index. Shuffle remaining so list is intact.
METHOD PUBLIC RemoveIndex : BOOL
VAR_INPUT
	Index : UDINT;
END_VAR
IF Index >= _Count THEN // invalid index request.
	RETURN;
END_IF

IF Index < _Count - 1 THEN // If Index = _Count -1, last two lines sufficient.

	MEMMOVE( 
		destAddr := ADR( List[Index] ), 
		srcAddr := ADR( List[Index + 1] ), 
		n := SIZEOF(List[0]) * (_Count - Index - 1)
	);
	
END_IF

List[_Count - 1] := 0; // default the "old" end of the list.
_Count := _Count - 1; // reduce count.
RemoveIndex := TRUE;
END_METHOD

// TRUE if successful and list item in sItem
METHOD PUBLIC TryGetIndex : BOOL
VAR_INPUT
	Index : PVOID;
END_VAR
VAR_IN_OUT
	Item : PVOID;
END_VAR
IF Index < _Count THEN
	TryGetIndex := TRUE;
	Item := List[Index];
ELSE
	Item := 0;
END_IF
END_METHOD

END_FUNCTION_BLOCK

// Utilities/Object Tracking/FB_LongStringList
// List of Strings.
FUNCTION_BLOCK FB_LongStringList
VAR
	List : ARRAY[ 0 .. GVL_List.LIST_SIZE - 1 ] OF LongString; // hold list
	_Count : UDINT := 0; // number of items.
END_VAR

// Add item to list. TRUE if successful. 
METHOD PUBLIC AddItem : BOOL
VAR_INPUT
	Item : LongString; // item to add.
END_VAR
IF _Count < GVL_List.LIST_SIZE THEN
	List[_Count] := Item; // list is zero indexed, so number of items points at next free space.
	_Count := _Count + 1; 
	AddItem := TRUE;
END_IF
END_METHOD

// Removes all list items
METHOD PUBLIC Clear
MEMSET(ADR(List[0]), 0, SIZEOF(List));
_Count := 0;
END_METHOD

// TRUE if Item is in FB_List.
METHOD PUBLIC Contains : BOOL
VAR_INPUT
	Item : LongString; // Item to check.
END_VAR
Contains := FindIndex(Item) >= 0;
END_METHOD

// TRUE if supplied key part is in any entry
METHOD PUBLIC ContainsPartial : BOOL
VAR_INPUT
	PartialItem : LongString;
END_VAR
ContainsPartial := FindIndexPartialKey(PartialItem) >= 0;
END_METHOD

METHOD CopyList
VAR_IN_OUT
	ListToCopyTo : ARRAY[ 0 .. GVL_List.LIST_SIZE - 1 ] OF LongString; // hold list
END_VAR
ListToCopyTo := THIS^.List;
END_METHOD

METHOD CopyListAndClear
VAR_IN_OUT
	ListToCopyTo : ARRAY[ 0 .. GVL_List.LIST_SIZE - 1 ] OF LongString; // hold list
END_VAR
THIS^.CopyList( ListToCopyTo );
THIS^.Clear();
END_METHOD

{attribute 'monitoring' := 'call'}
// Number of items in list.
PROPERTY PUBLIC Count : UDINT
GET
Count := _Count;
END_GET
END_PROPERTY

METHOD PUBLIC FindIndex : INT
VAR_INPUT
	Item : LongString; // Item to check.
END_VAR
VAR
	i : UINT := 0;
END_VAR
FindIndex := -1;
i := 0;
WHILE ( (FindIndex < 0) AND (i < _Count) ) DO
	
	FindIndex := SEL(Item = List[i], FindIndex, TO_INT(i) ); // if it matches, return the position.
	i := i + 1;
	
END_WHILE
END_METHOD

// Find first index where list entry contains supplied key.
METHOD PUBLIC FindIndexPartialKey : INT
VAR_INPUT
	PartialKey : LongString; // Item to check.
END_VAR
VAR
	i : UINT := 0;
END_VAR
FindIndexPartialKey := -1;
i := 0;
WHILE ( (FindIndexPartialKey < 0) AND (i < _Count) ) DO
	
	IF FIND(List[i],PartialKey) > 0 THEN
		FindIndexPartialKey := TO_INT(i);
	END_IF

	i := i + 1;
	
END_WHILE
END_METHOD

// Return item in list at index position. Returns empty string if invalid index.
METHOD PUBLIC GetIndex : LongString
VAR_INPUT
	Index : UDINT;
END_VAR
THIS^.TryGetIndex(Index,  GetIndex);
END_METHOD

//Remove the specified index. Shuffle remaining so list is intact.
METHOD PUBLIC RemoveIndex : BOOL
VAR_INPUT
	Index : UDINT;
END_VAR
IF Index >= _Count THEN // invalid index request.
	RETURN;
END_IF

IF Index < _Count - 1 THEN // If Index = _Count -1, last two lines sufficient.

	MEMMOVE( 
		destAddr := ADR( List[Index] ), 
		srcAddr := ADR( List[Index + 1] ), 
		n := SIZEOF(List[0]) * (_Count - Index - 1)
	);
	
END_IF

RemoveIndex := TRUE;

List[_Count - 1] := ''; // default the "old" end of the list.
_Count := _Count - 1; // reduce count.
END_METHOD

// TRUE if successful and list item in sItem
METHOD PUBLIC TryGetIndex : BOOL
VAR_INPUT
	Index : UDINT;
END_VAR
VAR_IN_OUT
	Item : LongString;
END_VAR
IF Index < _Count THEN
	TryGetIndex := TRUE;
	Item := List[Index];
END_IF
END_METHOD

END_FUNCTION_BLOCK

// Utilities/Object Tracking/FB_UdintList
// List of UDINTs.
FUNCTION_BLOCK FB_UdintList
VAR
	List : ARRAY[ 0 .. GVL_List.LIST_SIZE - 1 ] OF UDINT; // hold list
	_Count : UDINT := 0; // number of items.
END_VAR

// Add item to list. TRUE if successful. 
METHOD PUBLIC AddItem : BOOL
VAR_INPUT
	Item : UDINT; // item to add.
END_VAR
IF _Count < GVL_List.LIST_SIZE THEN
	List[_Count] := Item; // list is zero indexed, so number of items points at next free space.
	_Count := _Count + 1; 
	AddItem := TRUE;
END_IF
END_METHOD

// Removes all list items
METHOD PUBLIC Clear
MEMSET(ADR(List[0]), 0, SIZEOF(List));
_Count := 0;
END_METHOD

// TRUE if sItem is in FB_List.
METHOD PUBLIC Contains : BOOL
VAR_INPUT
	Item : UDINT; // Item to check.
END_VAR
Contains := FindIndex(Item) >= 0;
END_METHOD

{attribute 'monitoring' := 'call'}
// Number of items in list.
PROPERTY PUBLIC Count : UDINT
GET
Count := _Count;
END_GET
END_PROPERTY

METHOD PUBLIC FindIndex : INT
VAR_INPUT
	Item : UDINT; // Item to check.
END_VAR
VAR
	i : UINT := 0;
END_VAR
FindIndex := -1;
i := 0;
WHILE ( (FindIndex < 0) AND (i < _Count) ) DO
	
	FindIndex := SEL(Item = List[i], FindIndex, TO_INT(i) ); // if it matches, return the position.
	i := i + 1;
	
END_WHILE
END_METHOD

// Return item in list at index position. Returns empty string if invalid index.
METHOD PUBLIC GetIndex : UDINT
VAR_INPUT
	Index : UDINT;
END_VAR
THIS^.TryGetIndex(Index,  GetIndex);
END_METHOD

//Remove the specified index. Shuffle remaining so list is intact.
METHOD PUBLIC RemoveIndex : BOOL
VAR_INPUT
	Index : UDINT;
END_VAR
IF Index >= _Count THEN // invalid index request.
	RETURN;
END_IF

IF Index < _Count - 1 THEN // If Index = _Count -1, last two lines sufficient.

	MEMMOVE( 
		destAddr := ADR( List[Index] ), 
		srcAddr := ADR( List[Index + 1] ), 
		n := SIZEOF(List[0]) * (_Count - Index - 1)
	);
	
END_IF

RemoveIndex := TRUE;

List[_Count - 1] := 0; // default the "old" end of the list.
_Count := _Count - 1; // reduce count.
END_METHOD

// TRUE if successful and list item in sItem
METHOD PUBLIC TryGetIndex : BOOL
VAR_INPUT
	Index : UDINT;
END_VAR
VAR_IN_OUT
	Item : UDINT;
END_VAR
IF Index < _Count THEN
	TryGetIndex := TRUE;
	Item := List[Index];
ELSE
	Item := 0;
END_IF
END_METHOD

END_FUNCTION_BLOCK

// Utilities/PI Controller/FB_I_Controller
FUNCTION_BLOCK FB_I_Controller
VAR_INPUT
	ProcessVariable 		: LREAL;
	Setpoint				: LREAL;
	Ki						: LREAL; // Resets per unitTime
	MaxIntegralComponent 	: LREAL := 1000; // max absolute value of Output
	MinIntegralComponent	: LREAL := -1000; // min abs value of output.
	Pause					: BOOL;	// pause integration
	Reset					: BOOL; // reset integration.
END_VAR
VAR_OUTPUT
	Term					: LREAL;
END_VAR                 	
VAR                     	
	_Ki 					: LREAL; // include cycle time.
	integralComponent		: LREAL;
	error 					: LREAL;
	task 					: T_Task;
END_VAR

// if block turned off, do nothing.
IF Ki <= 0 THEN
	Term := 0;
	RETURN;
END_IF

IF Reset THEN
	integralComponent := 0;
ELSIF Pause THEN
	RETURN;
END_IF

// get gain with scan time.
_Ki := Ki * task.CycleTimeInSecs;

// get this error.
error := Setpoint - ProcessVariable  ;

// sum errors (gains included)
integralComponent := integralComponent + _Ki * error;

// clamp output, and reverse engineer integral accordingly.
IF integralComponent > MaxIntegralComponent THEN
	integralComponent := MaxIntegralComponent;
ELSIF integralComponent < MinIntegralComponent THEN
	integralComponent := MinIntegralComponent;
END_IF

// derive integral output.
Term := integralComponent;

END_FUNCTION_BLOCK

// Utilities/PI Controller/FB_P_Control
FUNCTION_BLOCK FB_P_Control
VAR_INPUT
	ProcessVariable : LREAL;
	Setpoint 		: LREAL;
	Kp 				: LREAL;
END_VAR         	
VAR_OUTPUT      	
	Term 			: LREAL;
END_VAR

Term := (Setpoint - ProcessVariable) * Kp;

END_FUNCTION_BLOCK

// Utilities/PI Controller/FB_PI_Controller
FUNCTION_BLOCK FB_PI_Controller
VAR_INPUT
	Reset				: BOOL; // Reset integral component
	ProcessVariable 	: LREAL;
	Setpoint			: LREAL;
	Kp					: LREAL;
	IntegralConstant 	: LREAL; // Repeats per minute
	RepeatsPerMinute	: BOOL := TRUE; // if false, repeats per second.
	MaxLoopOutput		: LREAL;
	MinLoopOutput		: LREAL;
	Bias				: LREAL;
END_VAR
VAR_OUTPUT
	Output 	: LREAL;
END_VAR
VAR
	p 		: FB_P_Control;
	i 		: FB_I_Controller;
	preClampedOutput : LREAL;
END_VAR

p(
	ProcessVariable:= ProcessVariable, 
	Setpoint:= Setpoint, 
	Kp:= Kp 
);

i(
	ProcessVariable := ProcessVariable, 
	Setpoint := Setpoint, 
	Ki	:= IntegralConstant / SEL(RepeatsPerMinute, 1, 60) , // normalising to repeats per minute. FB_I_COntroller block works in repeats per second natively.
	Pause := 
		( ( preClampedOutput > MaxLoopOutput ) AND ( ProcessVariable < Setpoint ) )
			OR 
		( ( preClampedOutput < MinLoopOutput ) AND ( ProcessVariable > Setpoint ) ),
	Reset := Reset
);

// caclculate output
preClampedOutput := p.Term + i.Term + Bias;
Output := LIMIT( MinLoopOutput, preClampedOutput, MaxLoopOutput ); // clamp the output

END_FUNCTION_BLOCK

// Utilities/String/Large Concats/F_ClearLarge
FUNCTION F_ClearLarge 
VAR_IN_OUT CONSTANT
	stringToClear 	: LongString;
END_VAR

MEMSET(ADR(stringToClear), 16#0, sizeof(stringToClear));

END_FUNCTION

// Utilities/String/Large Concats/F_Concat3_Large
FUNCTION F_Concat3_Large : LongString;
VAR_IN_OUT CONSTANT
	StringOne 	: LongString;
	StringTwo	: LongString;
	StringThree	: LongString;
END_VAR
VAR
	str : LongString;
END_VAR

str := F_ConcatLarge( StringTwo, StringThree );

F_Concat3_Large := 
	F_ConcatLarge(
		StringOne, 
		str
	);

END_FUNCTION

// Utilities/String/Large Concats/F_ConcatLarge
FUNCTION F_ConcatLarge : LongString
VAR_IN_OUT CONSTANT
	StringOne 	: LongString;
	StringTwo	: LongString;
END_VAR
VAR
	i, sizeToCpy, teminatingCharPos, maxLen : DINT;
	response : LongString;
END_VAR

maxLen := TO_DINT(StringsParams.MAX_STRING_LENGTH) - 1; // - 1 allows for terminating character in last position.

IF LEN(stringOne) + LEN(StringTwo) > maxLen THEN
	sizeToCpy := maxLen - LEN(StringTwo); //need room for the terminating character
	teminatingCharPos := maxLen; // this is the index position for utf-8 string as byte array

ELSE
	sizeToCpy := LEN(StringOne);
	teminatingCharPos := LEN(StringOne) + LEN(StringTwo);
	
END_IF

// copy strings into response
MEMCPY( ADR(response), ADR(StringOne), TO_UDINT(sizeToCpy) );
MEMCPY( ADR(response[sizeToCpy]), ADR(StringTwo), TO_UDINT( LEN(StringTwo) ) );

response[teminatingCharPos] := 16#0; // string terminating character
F_ConcatLarge := response;

END_FUNCTION

// Utilities/String/Large Concats/F_Concat4_Large
FUNCTION F_Concat4_Large : LongString
VAR_IN_OUT CONSTANT
	sOne 	: LongString;
	sTwo	: LongString;
	sThree	: LongString;
	sFour	: LongString;
END_VAR
VAR
	str : LongString;
END_VAR

str := F_Concat3_Large( sTwo, sThree, sFour);

F_Concat4_Large := 
	F_ConcatLarge(
		sOne,
		str
	);

END_FUNCTION

// Utilities/String/Large Concats/F_Concat5_Large
FUNCTION F_Concat5_Large : LongString
VAR_IN_OUT CONSTANT
	sOne : LongString;
	sTwo : LongString;
	sThree : LongString;
	sFour : LongString;
	sFive : LongString;
END_VAR
VAR
	str : LongString;
END_VAR

str := F_Concat4_Large( sTwo, sThree, sFour, sFive);
F_Concat5_Large := 
	F_ConcatLarge(
		sOne,
		str
	);

END_FUNCTION

// Utilities/String/Large Concats/F_Concat6_Large
FUNCTION F_Concat6_Large : LongString
VAR_IN_OUT CONSTANT
	sOne : LongString;
	sTwo : LongString;
	sThree : LongString;
	sFour : LongString;
	sFive : LongString;
	sSix : LongString;
END_VAR
VAR
	str : LongString;
END_VAR

str := F_Concat5_Large( sTwo, sThree, sFour, sFive, sSix);
F_Concat6_Large := 
	F_ConcatLarge(
		sOne,
		str
	);

END_FUNCTION

// Utilities/String/Large Concats/F_Concat7_Large
FUNCTION F_Concat7_Large : LongString
VAR_IN_OUT CONSTANT
	sOne : LongString;
	sTwo : LongString;
	sThree : LongString;
	sFour : LongString;
	sFive : LongString;
	sSix : LongString;
	sSeven : LongString;
END_VAR
VAR
	str : LongString;
END_VAR

str := F_Concat6_Large( sTwo, sThree, sFour, sFive, sSix, sSeven);
F_Concat7_Large := 
	F_ConcatLarge(
		sOne,
		str
	);

END_FUNCTION

// Utilities/String/F_Concat4
FUNCTION F_Concat4 : T_MaxString
VAR_INPUT
	sOne 	: STRING;
	sTwo	: STRING;
	sThree	: STRING;
	sFour	: STRING;
END_VAR

F_Concat4 := CONCAT(
					sOne,
					F_Concat3( sTwo, sThree, sFour )
				);

END_FUNCTION

// Utilities/String/F_Concat5
FUNCTION F_Concat5 : T_MaxString
VAR_INPUT
	sOne : STRING;
	sTwo : STRING;
	sThree : STRING;
	sFour : STRING;
	sFive : STRING;
END_VAR

F_Concat5 := CONCAT(
					sOne,
					F_Concat4( sTwo, sThree, sFour, sFive )
				);

END_FUNCTION

// Utilities/String/F_Concat6
FUNCTION F_Concat6 : T_MaxString
VAR_INPUT
	sOne : STRING;
	sTwo : STRING;
	sThree : STRING;
	sFour : STRING;
	sFive : STRING;
	sSix : STRING;
END_VAR

F_Concat6 := CONCAT(
					sOne,
					F_Concat5( sTwo, sThree, sFour, sFive, sSix )
				);

END_FUNCTION

// Utilities/String/F_Concat7
FUNCTION F_Concat7 : T_MaxString
VAR_INPUT
	sOne : STRING;
	sTwo : STRING;
	sThree : STRING;
	sFour : STRING;
	sFive : STRING;
	sSix : STRING;
	sSeven : STRING;
END_VAR

F_Concat7 := CONCAT(
					sOne,
					F_Concat6( sTwo, sThree, sFour, sFive, sSix, sSeven )
				);

END_FUNCTION

// Utilities/String/F_StringToTarg
FUNCTION F_StringToTarg
VAR_INPUT
	StringToConvert : T_MaxString;
END_VAR
VAR_IN_OUT
	Targ : T_ARG;
END_VAR
VAR
	b : POINTER TO BOOL;
	b8 : POINTER TO BYTE;
	w : POINTER TO WORD;
	dw : POINTER TO DWORD; 
	usi : POINTER TO USINT;
	si : POINTER TO SINT;
	ui : POINTER TO UINT;
	i : POINTER TO INT;
	udi : POINTER TO UDINT;
	di : POINTER TO DINT;
	str : POINTER TO STRING;
	re : POINTER TO REAL;
	lr : POINTER TO LREAL;
END_VAR

CASE Targ.eType OF
	
	E_ArgType.ARGTYPE_BOOL : 
		b := Targ.pData;
		b^ := TO_BOOL(StringToConvert);
		
	E_ArgType.ARGTYPE_BYTE : 
		b8 := Targ.pData;
		b8^ := TO_BYTE(StringToConvert);
		
	E_ArgType.ARGTYPE_WORD :
		w := Targ.pData;
		w^ := TO_WORD(StringToConvert);
	
	E_ArgType.ARGTYPE_DWORD :
		dw := Targ.pData;
		dw^ := TO_DWORD(StringToConvert);
		
	E_ArgType.ARGTYPE_USINT :
		usi := Targ.pData;
		usi^ := TO_USINT(StringToConvert);
		
	E_ArgType.ARGTYPE_SINT :
		si := Targ.pData;
		si^ := TO_SINT(StringToConvert);
	
	E_ArgType.ARGTYPE_UINT :
		ui := Targ.pData;
		ui^ := TO_UINT(StringToConvert);
		
	E_ArgType.ARGTYPE_INT :
		i := Targ.pData;
		i^ := TO_INT(StringToConvert);
		
	E_ArgType.ARGTYPE_UDINT :
		udi := Targ.pData;
		udi^ := TO_UDINT(StringToConvert);
		
	E_ArgType.ARGTYPE_DINT :
		di := Targ.pData;
		di^ := TO_DINT(StringToConvert);	
		
	E_ArgType.ARGTYPE_STRING :
		str := Targ.pData;
		str^ := TO_STRING(StringToConvert);	
		
	E_ArgType.ARGTYPE_REAL :
		re := Targ.pData;
		re^ := TO_REAL(StringToConvert);	
		
	E_ArgType.ARGTYPE_LREAL :
		lr := Targ.pData;
		lr^ := TO_LREAL(StringToConvert);	
	
	ELSE
		F_LogWarning(
			CONCAT(
				'Unsupported type in Targ for string conversion: ',
				TO_STRING(Targ.eType)
			)
		);
END_CASE

END_FUNCTION

// Utilities/String/F_TargToString
FUNCTION F_TargToString : T_MaxString
VAR_INPUT
	Targ : T_ARG;
END_VAR
VAR
	b : POINTER TO BOOL;
	b8 : POINTER TO BYTE;
	w : POINTER TO WORD;
	dw : POINTER TO DWORD; 
	usi : POINTER TO USINT;
	si : POINTER TO SINT;
	ui : POINTER TO UINT;
	i : POINTER TO INT;
	udi : POINTER TO UDINT;
	di : POINTER TO DINT;
	str : POINTER TO STRING;
	re : POINTER TO REAL;
	lr : POINTER TO LREAL;
END_VAR

CASE Targ.eType OF
	
	E_ArgType.ARGTYPE_BOOL : 
		b := Targ.pData;
		F_TargToString := TO_STRING(b^);
		
	E_ArgType.ARGTYPE_BYTE : 
		b8 := Targ.pData;
		F_TargToString := TO_STRING(b8^);
		
	E_ArgType.ARGTYPE_WORD :
		w := Targ.pData;
		F_TargToString := TO_STRING(w^);
	
	E_ArgType.ARGTYPE_DWORD :
		dw := Targ.pData;
		F_TargToString := TO_STRING(dw^);
		
	E_ArgType.ARGTYPE_USINT :
		usi := Targ.pData;
		F_TargToString := TO_STRING(usi^);
		
	E_ArgType.ARGTYPE_SINT :
		si := Targ.pData;
		F_TargToString := TO_STRING(si^);
	
	E_ArgType.ARGTYPE_UINT :
		ui := Targ.pData;
		F_TargToString := TO_STRING(ui^);
		
	E_ArgType.ARGTYPE_INT :
		i := Targ.pData;
		F_TargToString := TO_STRING(i^);
		
	E_ArgType.ARGTYPE_UDINT :
		udi := Targ.pData;
		F_TargToString := TO_STRING(udi^);
		
	E_ArgType.ARGTYPE_DINT :
		di := Targ.pData;
		F_TargToString := TO_STRING(di^);	
		
	E_ArgType.ARGTYPE_STRING :
		str := Targ.pData;
		F_TargToString := TO_STRING(str^);			
		
	E_ArgType.ARGTYPE_REAL :
		re := Targ.pData;
		F_TargToString := TO_STRING(re^);	
		
	E_ArgType.ARGTYPE_LREAL :
		lr := Targ.pData;
		F_TargToString := TO_STRING(lr^);	
	
	ELSE
		F_LogWarning(
			CONCAT(
				'Unsupported type in Targ for string conversion: ',
				TO_STRING(Targ.eType)
			)
		);
END_CASE

END_FUNCTION

// Utilities/Testing/FB_Assert
//A series of methods for use when testing functionality.
FUNCTION_BLOCK PUBLIC FB_Assert

METHOD FinishedTestingMsg
F_LogInfo('... Finished Testing');
END_METHOD

METHOD FINAL FloatsAreDifferent : BOOL
VAR_INPUT
	Float_1 : LREAL;
	Float_2 : LREAL;
	Precision : LREAL; // floating point precision.
	FailMsg : T_MaxString;
END_VAR
IF ABS(Float_1 - Float_2) <= Precision THEN
	F_LogError( 
		CONCAT('Assert.FloatsAreDifferent failed: ', FailMsg ) 
	);
ELSE
	FloatsAreDifferent := TRUE;
END_IF
END_METHOD

METHOD FINAL FloatsAreEqual : BOOL
VAR_INPUT
	Float_1 : LREAL;
	Float_2 : LREAL;
	Precision : LREAL; // floating point precision.
	FailMsg : T_MaxString;
END_VAR
IF ABS(Float_1 - Float_2) > Precision THEN
	F_LogError( 
		CONCAT('Assert.FloatsAreEqual failed: ', FailMsg ) 
	);
ELSE
	FloatsAreEqual := TRUE;
END_IF
END_METHOD

METHOD FINAL IsFalse : BOOL
VAR_INPUT
	Condition : BOOL;
	FailMsg : T_MaxString;
END_VAR
IF Condition THEN
	F_LogError( 
		CONCAT( 'Assert.IsFalse failed: ', FailMsg ) 
	);	
ELSE
	IsFalse := TRUE;
END_IF
END_METHOD

METHOD FINAL IsTrue : BOOL
VAR_INPUT
	Condition : BOOL;
	FailMsg : T_MaxString;
END_VAR
IF NOT Condition THEN
	F_LogError( 
		CONCAT( 'Assert.IsTrue failed: ', FailMsg ) 
	);
ELSE
	IsTrue := TRUE;
END_IF
END_METHOD

METHOD PUBLIC StartTestingMsg
F_LogInfo('Testing started...');
END_METHOD

END_FUNCTION_BLOCK

// Utilities/Testing/T_TestBase
FUNCTION_BLOCK T_TestBase EXTENDS T_NamedBase
VAR
	_done : BOOL;
	_testsPassed : BOOL;
	_reset : BOOL;
	_startTests : BOOL;
	_task : T_Task;
	_startTime : LINT; // ms
END_VAR

{attribute 'monitoring' := 'call'} PROPERTY Done : BOOL;
GET
Done := _done;
END_GET
SET
_done := Done;
END_SET
END_PROPERTY

{attribute 'monitoring' := 'call'} PROPERTY DonePulse : BOOL
GET
VAR_INST
	pulse : R_TRIG;
END_VAR
pulse( CLK := Done );
DonePulse := pulse.Q;
END_GET
END_PROPERTY

{attribute 'monitoring' := 'call'} PROPERTY nElapsedTimeInMs : LINT
GET
nElapsedTimeInMs := _task.DistributedClockTimeInMs - _startTime;
END_GET
END_PROPERTY

{attribute 'monitoring' := 'call'} PROPERTY Passed : BOOL;
GET
Passed := THIS^._testsPassed AND Done;
END_GET
END_PROPERTY

METHOD Reset
_reset := TRUE;
END_METHOD

METHOD Start
THIS^.Reset();
_startTests := TRUE;
END_METHOD

METHOD StartTimer
_task.SetToThisTask(); // which ever thread this is called on sets the timer.
_startTime := _task.DistributedClockTimeInMs;
END_METHOD

{attribute 'monitoring' := 'call'} PROPERTY tElapsedTimeInMs : TIME
GET
tElapsedTimeInMs := TO_TIME(nElapsedTimeInMs);
END_GET
END_PROPERTY

END_FUNCTION_BLOCK

// Utilities/Timers/T_Timer
FUNCTION_BLOCK T_Timer // a timer block. Will start timing as soon as T_Timer.Signal is present. 
VAR_INPUT
END_VAR
VAR
	task : T_Task;
	startTime : LINT; // ms
	_elapsedTimeInMs : LINT;
	_duration : LINT := 1;
	_signal : BOOL;
	_offSignal : BOOL;
END_VAR

{attribute 'monitoring' := 'call'} PROPERTY ElapsedTime : TIME // returns 0 if Signal = FALSE;
GET
ElapsedTime := LINT_TO_TIME( ElapsedTimeInMs );
END_GET
END_PROPERTY

{attribute 'monitoring' := 'call'} PROPERTY ElapsedTimeInMs : LINT // returns 0 if Signal = FALSE;
GET
ElapsedTimeInMs := 
	SEL(_signal, 0,  task.DistributedClockTimeInMs - startTime);
END_GET
END_PROPERTY

PROPERTY Q_Off : BOOL
GET
Q_Off := _offSignal AND_THEN
			( ( task.DistributedClockTimeInMs - startTime ) > _duration );
END_GET
END_PROPERTY

PROPERTY Q_On : BOOL
GET
Q_On := _signal AND_THEN
			( ( task.DistributedClockTimeInMs - startTime ) > _duration );
END_GET
END_PROPERTY

PROPERTY Q_PulseTrain : BOOL
GET
Q_PulseTrain := _signal AND_THEN
			( ( task.DistributedClockTimeInMs - startTime ) MOD _duration > ( _duration / 2 ) );
END_GET
END_PROPERTY

PROPERTY SetPeriod : TIME
GET
SetPeriod := LINT_TO_TIME( _duration );
END_GET
SET
_duration := MAX( TIME_TO_LINT( SetPeriod ), 1);
END_SET
END_PROPERTY

PROPERTY Signal : BOOL
GET
Signal := _signal;
END_GET
SET
IF Signal <> _signal THEN
	startTime := task.DistributedClockTimeInMs;
	_signal := Signal;
	_offSignal := NOT _signal;
END_IF
END_SET
END_PROPERTY

END_FUNCTION_BLOCK

// Utilities/Write persistent/T_WritePersistentData
/// default is port 851, every 10s.
FUNCTION_BLOCK T_WritePersistentData
VAR
	writePersistent: FB_WritePersistentData;
	writePeriod: TIME := TIME#10s0ms;
	adsPort: UINT := 851;
	writePersistTimer: TON;
END_VAR

// periodic force write of persistant variables.
writePersistTimer( IN := NOT writePersistTimer.Q, PT := writePeriod );
writePersistent( PORT:= adsPort, START := writePersistTimer.Q );

METHOD SetConfig : BOOL
VAR_INPUT
	/// How often to write data to persistent (default is 10S)/
	WritePeriod: TIME;
	/// which ads port (default is 851)
	AdsPort: UINT;
END_VAR
END_METHOD

END_FUNCTION_BLOCK

// Utilities/F_Gate
// return the bIn as passed. set the value to FALSE.
FUNCTION F_Gate : BOOL
VAR_IN_OUT
	bIn : BOOL;
END_VAR

F_Gate := bIn;
// reset if true. (below is equivalent of IF bIn THEN bIn := FALSE; END_IF)
bIn := FALSE;

END_FUNCTION
